SUBAPPLICATION SINT_TO_Q_NumericValue (* SINT-Wert (z.B. Schrittkettennummer) auf ein VT-Zahlenfeld (Q_NumericValue) anzeigen. Generisch, Object ID parametrierbar. *)
  (* Standard: 61499-2 *)
  (* Version 1.0, 2026-09-09, Franz Höpfinger, Meisterschulen am Ostbahnhof, Ausgelagert aus Uebung_039_sub_NumbAnzeig zur Wiederverwendung; u16ObjId zuvor fest importiert (OutputNumber_N1), jetzt als VarDeclaration parametrierbar. *)
  PACKAGE MyLib::sys;
  IMPORT isobus::UT::Q::const::IDs::ID_NULL;
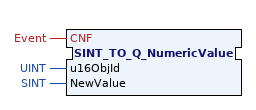
  EVENT_INPUT
    CNF;
  END_EVENT
  VAR_INPUT
    u16ObjId : UINT := ID_NULL; (* Object ID *)
    NewValue : SINT;
  END_VAR
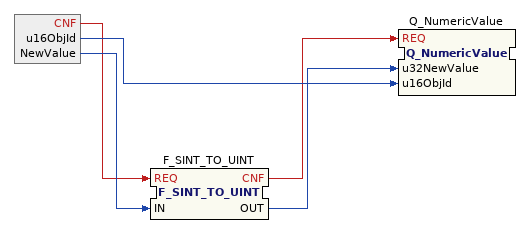
  FBS
    F_SINT_TO_UINT : iec61131::conversion::F_SINT_TO_UINT;
    Q_NumericValue : isobus::UT::Q::Q_NumericValue;
  END_FBS
  EVENT_CONNECTIONS
    F_SINT_TO_UINT.CNF TO Q_NumericValue.REQ;
    CNF TO F_SINT_TO_UINT.REQ;
  END_CONNECTIONS
  DATA_CONNECTIONS
    F_SINT_TO_UINT.OUT TO Q_NumericValue.u32NewValue;
    NewValue TO F_SINT_TO_UINT.IN;
    u16ObjId TO Q_NumericValue.u16ObjId;
  END_CONNECTIONS
END_SUBAPPLICATION
